PROGRAM MAIN
VAR
	hueClient:	FB_IotHttpClient := (sHostName := '192.168.1.53', bKeepAlive := TRUE, tConnectionTimeout := T#5S);
	hueRequest:	FB_IotHttpRequest;
	
	jsonParser:	FB_JSONDomParser;
	jsonWriter:	FB_JsonSaxWriter;
	jsonDoc:	SJsonValue;
	jsonLight1:	SJsonValue;
	jsonLight1Status:	SJsonValue;
	jsonLightOn:	SJsonValue;
	jsonLightBrightness:	SJsonValue;
	jsonLightHue:	SJsonValue;
	jsonLightSat:	SJsonValue;
	
	Light1On:	BOOL;
	Light1Brightness:	DINT;
	Light1Hue:	DINT;
	Light1Sat:	DINT;
	
	sContent:	STRING(2048);
	sCommand:	STRING;
	
	bGetLights:	BOOL;
	nState:	INT;
	apiKey:	STRING := 'S9U3UinAsoFCoKTF8iFRW-jewXsCee9qjEFFEYHf';
	tempURI:	STRING;
	
	bLightSetOn	AT %I*:	BOOL;
	nLightSetBri:	INT;
	nLightSetHue	AT %I*:	UINT;
	nLightSetHueAuto:	UDINT;
	nLightSetSat:	INT;
	
	Pot1	AT %I*:	INT;
	Pot2	AT %I*: INT;
	
	Timer:	TON;
	rtSend:	R_TRIG;
	bStep: BOOL;
	bConnected: BOOL;
	bRun: BOOL;
	nErrorCount:	UDINT;
END_VAR

nLightSetBri := F_Scale(Pot1);
nLightSetSat := F_Scale(Pot2);

IF NOT hueClient.bConfigured THEN
	hueClient.nHostPort := 80;
	hueClient.stTLS.bNoServerCertCheck := FALSE;
END_IF

IF bGetLights THEN
	bGetLights := FALSE;
	nState := 10;
END_IF

Timer( IN := NOT Timer.Q, PT := T#100MS);
rtSend(CLK := Timer.Q);

IF hueClient.bConnected THEN
	bConnected := TRUE;
END_IF

CASE nState OF
	0:
		IF (bStep OR bRun) AND hueClient.bConfigured THEN
			bStep := FALSE;
			nState := nState + 1;
		END_IF
		
	1:
		jsonWriter.StartObject();
		jsonWriter.AddKey('on');
		jsonWriter.AddBool(bLightSetOn);
		jsonWriter.AddKey('sat');
		jsonWriter.AddUdint(nLightSetSat);
		jsonWriter.AddKey('bri');
		jsonWriter.AddUdint(nLightSetBri);
		jsonWriter.AddKey('hue');
		jsonWriter.AddUdint(nLightSetHueAuto);
		jsonWriter.EndObject();
		sCommand := jsonWriter.GetDocument();
		jsonWriter.ResetDocument();
		nState := nState + 1;
		
	2:
		tempURI := CONCAT(CONCAT('/api/', apiKey), '/lights/1/state');
		IF hueRequest.SendRequest(sUri := tempURI,
									fbClient := hueClient,
									eRequestType := ETcIotHttpRequestType.HTTP_PUT,
									pContent := ADR(sCommand),
									nContentSize := SIZEOF(sCommand),
									fbHeader := 0) THEN
			nState := nState + 1;
		END_IF
		
	3:
		IF NOT hueRequest.bBusy THEN
			IF hueRequest.bError THEN
				nErrorCount := nErrorCount + 1;
				nState := 1;
			ELSE
				IF (bStep OR bRun) THEN
					bStep := FALSE;
					nState := nState + 1;
				END_IF
			END_IF
		END_IF
		
	4:
		hueClient.Disconnect();
		IF (bStep OR bRun) AND NOT hueClient.bConnected THEN
			bStep := FALSE;
			nState := nState + 1;
		END_IF
		
	5:
		IF (bStep OR bRun) THEN
			bStep := FALSE;
			nState := 0;
		END_IF
		
END_CASE

(*CASE nState OF
	0: //IDLE
		IF rtSend.Q THEN
			nState := nState + 1;
		END_IF
	
	1:
		nLightSetHueAuto := nLightSetHueAuto + 5000;
		IF nLightSetHueAuto = 65000 THEN
			nLightSetHueAuto := 0;
		END_IF
		jsonWriter.StartObject();
		jsonWriter.AddKey('on');
		jsonWriter.AddBool(bLightSetOn);
		jsonWriter.AddKey('sat');
		jsonWriter.AddUdint(nLightSetSat);
		jsonWriter.AddKey('bri');
		jsonWriter.AddUdint(nLightSetBri);
		jsonWriter.AddKey('hue');
		jsonWriter.AddUdint(nLightSetHueAuto);
		jsonWriter.EndObject();
		sCommand := jsonWriter.GetDocument();
		jsonWriter.ResetDocument();
		nState := nState + 1;

	2:
		tempURI := CONCAT(CONCAT('/api/', apiKey), '/lights/1/state');
		IF hueRequest.SendRequest(sUri := tempURI,
									fbClient := hueClient,
									eRequestType := ETcIotHttpRequestType.HTTP_PUT,
									pContent := ADR(sCommand),
									nContentSize := SIZEOF(sCommand),
									fbHeader := 0) THEN
			nState := nState + 1;
		END_IF
		
	3:
		IF NOT hueRequest.bBusy THEN
			IF hueRequest.bError THEN
				nState := 500;
			ELSE
				nState := 10;
			END_IF
		END_IF
	
	10:	//Get Light Status
		tempURI := CONCAT(CONCAT('/api/', apiKey),'/lights');
		IF hueRequest.SendRequest(sUri := tempURI,
								fbClient := hueClient,
								eRequestType := ETciotHttpRequestType.HTTP_GET,
								0, 0, 0) THEN
			nState := nState + 1;
		END_IF
		
	11:
		IF NOT hueRequest.bBusy THEN
			IF hueRequest.bError THEN
				nState := 500;
			ELSE
				hueRequest.GetContent(pContent := ADR(sContent),
										nContentSize := SIZEOF(sContent),
										bSetNullTermination := TRUE);
				IF hueRequest.nStatusCode >= 200 AND hueRequest.nStatusCode < 300 THEN
					jsonDoc := hueRequest.GetJsonDomContent(jsonParser);
					jsonLight1 := jsonParser.FindMember(jsonDoc, '1');
					jsonLight1Status := jsonParser.FindMember(jsonLight1, 'state');
					jsonLightOn := jsonParser.FindMember(jsonLight1Status, 'on');
					jsonLightBrightness := jsonParser.FindMember(jsonLight1Status, 'bri');
					jsonLightHue := jsonParser.FindMember(jsonLight1Status, 'hue');
					jsonLightSat := jsonParser.FindMember(jsonLight1Status, 'sat');
					
					Light1On := jsonParser.GetBool(jsonLightOn);
					Light1Brightness := jsonParser.GetInt(jsonLightBrightness);
					Light1Hue := jsonParser.GetInt(jsonLightHue);
					Light1Sat := jsonParser.GetInt(jsonLightSat);
				END_IF
				nState := 0;
			END_IF
		END_IF
		
END_CASE*)

hueClient.Execute();

END_PROGRAM

(* stored: Version 1.1.0.1, ProductVersion 3.1.4024.11
   POU MAIN: Id {ecb56928-c082-44ca-97ca-1d3ddd69cd92}, SpecialFunc None *)
